FUNCTION_BLOCK EL_StopperArm (* StopperArm: commands -> outputs in timed phases (break before make); one holder at a time; all off when the module aborts; inputs -> state channel *)
  (* Standard: 61499-2 *)
  (* Version 0.1, 2026-09-28, Project contributors, AAU Smart Production Lab *)
  PACKAGE stoppering;
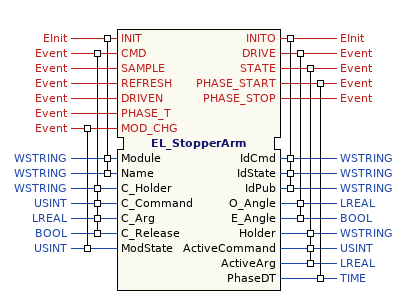
  EVENT_INPUT
    INIT : EInit WITH Module, Name;
    CMD WITH C_Holder, C_Command, C_Arg, C_Release;
    SAMPLE;
    REFRESH;
    DRIVEN;
    PHASE_T;
    MOD_CHG WITH ModState;
  END_EVENT
  EVENT_OUTPUT
    INITO : EInit WITH IdCmd, IdState, IdPub;
    DRIVE WITH O_Angle, E_Angle;
    STATE WITH Holder, ActiveCommand, ActiveArg;
    PHASE_START WITH PhaseDT;
    PHASE_STOP;
  END_EVENT
  VAR_INPUT
    Module : WSTRING;
    Name : WSTRING;
    C_Holder : WSTRING;
    C_Command : USINT;
    C_Arg : LREAL;
    C_Release : BOOL;
    ModState : USINT;
  END_VAR
  VAR_OUTPUT
    IdCmd : WSTRING;
    IdState : WSTRING;
    IdPub : WSTRING;
    O_Angle : LREAL;
    E_Angle : BOOL;
    Holder : WSTRING;
    ActiveCommand : USINT;
    ActiveArg : LREAL;
    PhaseDT : TIME;
  END_VAR
  VAR
    Command : USINT;
    Phase : USINT;
    Arg : LREAL;
    Changed : BOOL;
    Timed : BOOL;
    Publish : BOOL;
    Beat : USINT;
    LastHolder : WSTRING;
    Pending : BOOL;
    AbortPending : BOOL;
    N_Angle : LREAL;
    NE_Angle : BOOL;
  END_VAR
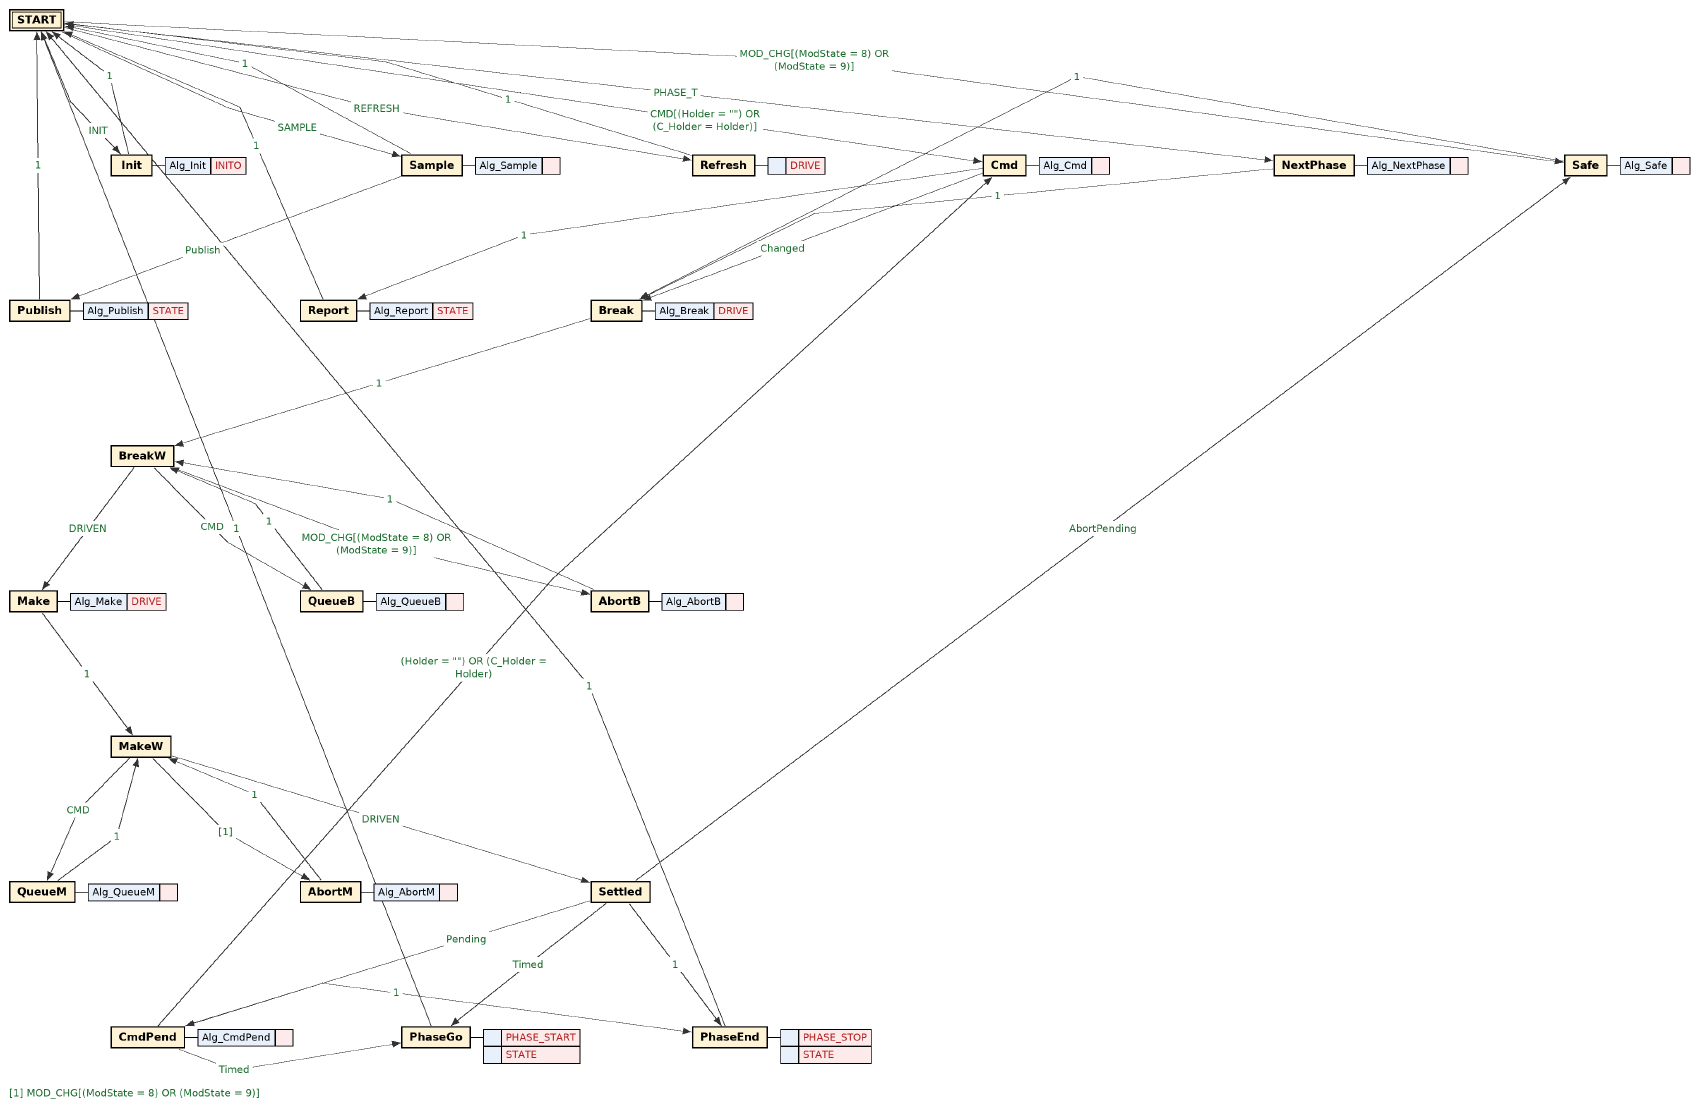
  EC_STATES
    START;
    Init : Alg_Init -> INITO;
    Sample : Alg_Sample;
    Publish : Alg_Publish -> STATE;
    Refresh : -> DRIVE;
    Cmd : Alg_Cmd;
    Report : Alg_Report -> STATE;
    NextPhase : Alg_NextPhase;
    Safe : Alg_Safe;
    Break : Alg_Break -> DRIVE;
    Make : Alg_Make -> DRIVE;
    BreakW;
    MakeW;
    QueueB : Alg_QueueB;
    AbortB : Alg_AbortB;
    QueueM : Alg_QueueM;
    AbortM : Alg_AbortM;
    CmdPend : Alg_CmdPend;
    Settled;
    PhaseGo : -> PHASE_START, -> STATE;
    PhaseEnd : -> PHASE_STOP, -> STATE;
  END_STATES
  EC_TRANSITIONS
    START TO Init := INIT;
    START TO Sample := SAMPLE;
    START TO Refresh := REFRESH;
    START TO Cmd := CMD[(Holder = "") OR (C_Holder = Holder)];
    START TO NextPhase := PHASE_T;
    START TO Safe := MOD_CHG[(ModState = 8) OR (ModState = 9)];
    Init TO START := 1;
    Sample TO Publish := Publish;
    Sample TO START := 1;
    Publish TO START := 1;
    Refresh TO START := 1;
    Cmd TO Break := Changed;
    Cmd TO Report := 1;
    Report TO START := 1;
    NextPhase TO Break := 1;
    Safe TO Break := 1;
    Break TO BreakW := 1;
    BreakW TO Make := DRIVEN;
    Make TO MakeW := 1;
    MakeW TO Settled := DRIVEN;
    BreakW TO QueueB := CMD;
    BreakW TO AbortB := MOD_CHG[(ModState = 8) OR (ModState = 9)];
    QueueB TO BreakW := 1;
    AbortB TO BreakW := 1;
    MakeW TO QueueM := CMD;
    MakeW TO AbortM := MOD_CHG[(ModState = 8) OR (ModState = 9)];
    QueueM TO MakeW := 1;
    AbortM TO MakeW := 1;
    Settled TO Safe := AbortPending;
    Settled TO CmdPend := Pending;
    CmdPend TO Cmd := (Holder = "") OR (C_Holder = Holder);
    CmdPend TO PhaseGo := Timed;
    CmdPend TO PhaseEnd := 1;
    Settled TO PhaseGo := Timed;
    Settled TO PhaseEnd := 1;
    PhaseGo TO START := 1;
    PhaseEnd TO START := 1;
  END_TRANSITIONS
  ALGORITHM Alg_Init IN ST:
IdCmd := CONCAT(CONCAT(CONCAT(CONCAT("loc[", Module), "/"), Name), "/cmd]");
IdState := CONCAT(CONCAT(CONCAT(CONCAT("loc[", Module), "/"), Name), "/state]");
IdPub := "";
  END_ALGORITHM
  ALGORITHM Alg_Sample IN ST:
Publish := (Holder <> LastHolder) OR (Beat >= 20);
Beat := Beat + 1;
ActiveCommand := Command;
ActiveArg := Arg;
  END_ALGORITHM
  ALGORITHM Alg_Publish IN ST:
LastHolder := Holder;
Beat := 0;
  END_ALGORITHM
  ALGORITHM Alg_Cmd IN ST:
Holder := C_Holder;
Changed := (C_Command <> 255) AND ((C_Command <> Command) OR (C_Arg <> Arg));
IF Changed THEN
  Command := C_Command;
  Phase := 0;
  Arg := C_Arg;
END_IF;
IF C_Release THEN
  Holder := "";
END_IF;
  END_ALGORITHM
  ALGORITHM Alg_Report IN ST:
LastHolder := Holder;
Beat := 0;
  END_ALGORITHM
  ALGORITHM Alg_NextPhase IN ST:
Phase := Phase + 1;
  END_ALGORITHM
  ALGORITHM Alg_Safe IN ST:
Command := 0;
Phase := 0;
Holder := "";
AbortPending := FALSE;
  END_ALGORITHM
  ALGORITHM Alg_Break IN ST:
N_Angle := 0.0;
NE_Angle := FALSE;
Timed := FALSE;
PhaseDT := T#0ms;
IF Command = 1 THEN
  N_Angle := Arg;
  NE_Angle := TRUE;
END_IF;
  END_ALGORITHM
  ALGORITHM Alg_Make IN ST:
O_Angle := N_Angle;
E_Angle := NE_Angle;
  END_ALGORITHM
  ALGORITHM Alg_QueueB IN ST:
Pending := TRUE;
  END_ALGORITHM
  ALGORITHM Alg_AbortB IN ST:
AbortPending := TRUE;
  END_ALGORITHM
  ALGORITHM Alg_QueueM IN ST:
Pending := TRUE;
  END_ALGORITHM
  ALGORITHM Alg_AbortM IN ST:
AbortPending := TRUE;
  END_ALGORITHM
  ALGORITHM Alg_CmdPend IN ST:
Pending := FALSE;
  END_ALGORITHM
END_FUNCTION_BLOCK
